// TwinCAT 3 PLC project Tc3EventLoggerListener
// Title: Tc3EventLoggerListener
// Company: tchaxx
// Author: densogiaichned
// ProjectVersion: 0.0.1.0
// Description: Example how to use TC3 EventLogger
// ProgramVersion: 3.1.4024.0
// libraries:
//   Tc2_Standard, * (Beckhoff Automation GmbH)
//   Tc2_System, * (Beckhoff Automation GmbH)
//   Tc2_Utilities, * (Beckhoff Automation GmbH)
//   Tc3_EventLogger, * (Beckhoff Automation GmbH)
//   Tc3_Module, * (Beckhoff Automation GmbH)
//   TcUnit, * (www.tcunit.org)
// project tree:
//   DUTs/ E_EventLoggerListenerState.TcTLEO, E_LanguageId.TcTLEO, ST_LoggedEvent.TcDUT, ST_RequestEventTexts.TcDUT, T_LoggedEvents.TcDUT, T_RequestEventTexts.TcDUT
//   GVLs/ Param_EventLoggerListener.TcGVL
//   ITFs/ I_LoggedEventsSort.TcIO
//   / PlcTask.TcTTO, PlcTaskUnitTest.TcTTO
//   POUs/ FB_EventLoggerListenerImpl.TcPOU, FB_LoggedEventsSortAscending.TcPOU, FB_LoggedEventsSortDescending.TcPOU, MAIN.TcPOU
//   TESTs/ FB_LoggedEventsSortDescending_Tests.TcPOU, PRG_UnitTests.TcPOU
// real-time tasks:
//   TASK PlcTask: cycle T#10ms, priority 20, ADS port 350
//   TASK PlcTaskUnitTest: cycle T#10ms, priority 1, ADS port 351

CONFIGURATION Tc3EventLoggerListener
    RESOURCE PLC ON TwinCAT3
        TASK PlcTask(INTERVAL := T#10ms, PRIORITY := 20);
        TASK PlcTaskUnitTest(INTERVAL := T#10ms, PRIORITY := 1);
        PROGRAM MAIN WITH PlcTask : MAIN;
        PROGRAM PRG_UnitTests WITH PlcTaskUnitTest : PRG_UnitTests;
    END_RESOURCE
END_CONFIGURATION

// ---- DUTs/E_EventLoggerListenerState.TcTLEO
{attribute 'qualified_only'}
{attribute 'strict'}
{attribute 'to_string'}
TYPE E_EventLoggerListenerState :
(	 
	eIdle := 0,
	eInit:= 1, 
	eListening:= 10, 
	eRetrieveTexts:= 20,
	eSortEvents := 30,
	eDone := 100,
	eError := -1
);
END_TYPE
//  eError = '-1'

// ---- DUTs/E_LanguageId.TcTLEO
{attribute 'qualified_only'}
{attribute 'strict'}
TYPE E_LanguageId :
(
	ar_SA := 1025 , // Arabic - Saudi Arabia
	bg_BG := 1026 , // Bulgarian
	ca_ES := 1027 , // Catalan
	zh_TW := 1028 , // Chinese - Taiwan
	cs_CZ := 1029 , // Czech
	da_DK := 1030 , // Danish
	de_DE := 1031 , // German - Germany
	el_GR := 1032 , // Greek
	en_US := 1033 , // English - United States
	es_ES := 1034 , // Spanish - Spain (Traditional Sort)
	fi_FI := 1035 , // Finnish
	fr_FR := 1036 , // French - France
	he_IL := 1037 , // Hebrew
	hu_HU := 1038 , // Hungarian
	is_IS := 1039 , // Icelandic
	it_IT := 1040 , // Italian - Italy
	ja_JP := 1041 , // Japanese
	ko_KR := 1042 , // Korean
	nl_NL := 1043 , // Dutch - Netherlands
	nb_NO := 1044 , // Norwegian (Bokmål)
	pl_PL := 1045 , // Polish
	pt_BR := 1046 , // Portuguese - Brazil
	rm_CH := 1047 , // Rhaeto-Romanic
	ro_RO := 1048 , // Romanian
	ru_RU := 1049 , // Russian
	hr_HR := 1050 , // Croatian
	sk_SK := 1051 , // Slovak
	sq_AL := 1052 , // Albanian - Albania
	sv_SE := 1053 , // Swedish
	th_TH := 1054 , // Thai
	tr_TR := 1055 , // Turkish
	ur_PK := 1056 , // Urdu - Pakistan
	id_ID := 1057 , // Indonesian
	uk_UA := 1058 , // Ukrainian
	be_BY := 1059 , // Belarusian
	sl_SI := 1060 , // Slovenian
	et_EE := 1061 , // Estonian
	lv_LV := 1062 , // Latvian
	lt_LT := 1063 , // Lithuanian
	tg_Cyrl_TJ := 1064 , // Tajik
	fa_IR := 1065 , // Persian
	vi_VN := 1066 , // Vietnamese
	hy_AM := 1067 , // Armenian - Armenia
	az_Latn_AZ := 1068 , // Azerbaijani (Latin)
	eu_ES := 1069 , // Basque
	wen_DE := 1070 , // Sorbian
	mk_MK := 1071 , // North Macedonian
	st_ZA := 1072 , // Sutu
	ts_ZA := 1073 , // Tsonga
	tn_ZA := 1074 , // Tswana
	ven_ZA := 1075 , // Venda
	xh_ZA := 1076 , // Xhosa
	zu_ZA := 1077 , // Zulu
	af_ZA := 1078 , // Afrikaans - South Africa
	ka_GE := 1079 , // Georgian
	fo_FO := 1080 , // Faroese
	hi_IN := 1081 , // Hindi
	mt_MT := 1082 , // Maltese
	se_NO := 1083 , // Sami
	gd_GB := 1084 , // Scottish Gaelic
	yi := 1085 , // Yiddish
	ms_MY := 1086 , // Malay - Malaysia
	kk_KZ := 1087 , // Kazakh
	ky_KG := 1088 , // Kyrgyz (Cyrillic)
	sw_KE := 1089 , // Swahili
	tk_TM := 1090 , // Turkmen
	uz_Latn_UZ := 1091 , // Uzbek (Latin)
	tt_RU := 1092 , // Tatar
	bn_IN := 1093 , // Bengali (India)
	pa_IN := 1094 , // Punjabi
	gu_IN := 1095 , // Gujarati
	or_IN := 1096 , // Odia
	ta_IN := 1097 , // Tamil
	te_IN := 1098 , // Telugu
	kn_IN := 1099 , // Kannada
	ml_IN := 1100 , // Malayalam
	as_IN := 1101 , // Assamese
	mr_IN := 1102 , // Marathi
	sa_IN := 1103 , // Sanskrit
	mn_MN := 1104 , // Mongolian (Cyrillic)
	bo_CN := 1105 , // Tibetan - People's Republic of China
	cy_GB := 1106 , // Welsh
	km_KH := 1107 , // Khmer
	lo_LA := 1108 , // Lao
	my_MM := 1109 , // Burmese
	gl_ES := 1110 , // Galician
	kok_IN := 1111 , // Konkani
	mni := 1112 , // Manipuri
	sd_IN := 1113 , // Sindhi - India
	syr_SY := 1114 , // Syriac
	si_LK := 1115 , // Sinhalese - Sri Lanka
	chr_US := 1116 , // Cherokee - United States
	iu_Cans_CA := 1117 , // Inuktitut
	am_ET := 1118 , // Amharic - Ethiopia
	tmz := 1119 , // Tamazight (Arabic)
	ks_Arab_IN := 1120 , // Kashmiri (Arabic)
	ne_NP := 1121 , // Nepali
	fy_NL := 1122 , // Frisian - Netherlands
	ps_AF := 1123 , // Pashto
	fil_PH := 1124 , // Filipino
	dv_MV := 1125 , // Divehi
	bin_NG := 1126 , // Edo
	fuv_NG := 1127 , // Fulfulde - Nigeria
	ha_Latn_NG := 1128 , // Hausa - Nigeria
	ibb_NG := 1129 , // Ibibio - Nigeria
	yo_NG := 1130 , // Yoruba
	quz_BO := 1131 , // Quecha - Bolivia
	nso_ZA := 1132 , // Sepedi
	ig_NG := 1136 , // Igbo - Nigeria
	kr_NG := 1137 , // Kanuri - Nigeria
	gaz_ET := 1138 , // Oromo
	ti_ER := 1139 , // Tigrigna - Ethiopia
	gn_PY := 1140 , // Guarani - Paraguay
	haw_US := 1141 , // Hawaiian - United States
	la := 1142 , // Latin
	so_SO := 1143 , // Somali
	ii_CN := 1144 , // Yi
	pap_AN := 1145 , // Papiamentu
	ug_Arab_CN := 1152 , // Uighur - China
	mi_NZ := 1153 , // Maori - New Zealand
	ar_IQ := 2049 , // Arabic - Iraq
	zh_CN := 2052 , // Chinese - People's Republic of China
	de_CH := 2055 , // German - Switzerland
	en_GB := 2057 , // English - United Kingdom
	es_MX := 2058 , // Spanish - Mexico
	fr_BE := 2060 , // French - Belgium
	it_CH := 2064 , // Italian - Switzerland
	nl_BE := 2067 , // Dutch - Belgium
	nn_NO := 2068 , // Norwegian (Nynorsk)
	pt_PT := 2070 , // Portuguese - Portugal
	ro_MD := 2072 , // Romanian - Moldova
	ru_MD := 2073 , // Russian - Moldava
	sr_Latn_CS := 2074 , // Serbian (Latin)
	sv_FI := 2077 , // Swedish - Finland
	ur_IN := 2080 , // Urdu - India
	az_Cyrl_AZ := 2092 , // Azerbaijani (Cyrillic)
	ga_IE := 2108 , // Irish
	ms_BN := 2110 , // Malay - Brunei Darussalam
	uz_Cyrl_UZ := 2115 , // Uzbek (Cyrillic)
	bn_BD := 2117 , // Bangla
	pa_PK := 2118 , // Punjabi (Pakistan)
	mn_Mong_CN := 2128 , // Mongolian (Mongolian)
	bo_BT := 2129 , // Tibetan - Bhutan
	sd_PK := 2137 , // Sindhi - Pakistan
	tzm_Latn_DZ := 2143 , // Tamazight (Latin)
	ks_Deva_IN := 2144 , // Kashmiri (Devanagari)
	ne_IN := 2145 , // Nepali - India
	quz_EC := 2155 , // Quecha - Ecuador
	ti_ET := 2163 , // Tigrigna - Eritrea
	ar_EG := 3073 , // Arabic - Egypt
	zh_HK := 3076 , // Chinese - Hong Kong SAR
	de_AT := 3079 , // German - Austria
	en_AU := 3081 , // English - Australia
	es_ES2 := 3082 , // Spanish - Spain (Modern Sort)
	fr_CA := 3084 , // French - Canada
	sr_Cyrl_CS := 3098 , // Serbian (Cyrillic)
	quz_PE := 3179 , // Quecha - Peru
	ar_LY := 4097 , // Arabic - Libya
	zh_SG := 4100 , // Chinese - Singapore
	de_LU := 4103 , // German - Luxembourg
	en_CA := 4105 , // English - Canada
	es_GT := 4106 , // Spanish - Guatemala
	fr_CH := 4108 , // French - Switzerland
	hr_BA := 4122 , // Croatian (Bosnia/Herzegovina)
	ar_DZ := 5121 , // Arabic - Algeria
	zh_MO := 5124 , // Chinese - Macao SAR
	de_LI := 5127 , // German - Liechtenstein
	en_NZ := 5129 , // English - New Zealand
	es_CR := 5130 , // Spanish - Costa Rica
	fr_LU := 5132 , // French - Luxembourg
	bs_Latn_BA := 5146 , // Bosnian (Bosnia/Herzegovina)
	ar_MO := 6145 , // Arabic - Morocco
	en_IE := 6153 , // English - Ireland
	es_PA := 6154 , // Spanish - Panama
	fr_MC := 6156 , // French - Monaco
	ar_TN := 7169 , // Arabic - Tunisia
	en_ZA := 7177 , // English - South Africa
	es_DO := 7178 , // Spanish - Dominican Republic
	ar_OM := 7180 , // French - West Indies,fr-Arabic - Oman
	en_JM := 8201 , // English - Jamaica
	es_VE := 8202 , // Spanish - Venezuela
	fr_RE := 8204 , // French - Reunion
	ar_YE := 9217 , // Arabic - Yemen
	es_CO := 9225 , // English - Caribbean,en-Spanish - Colombia
	fr_CG := 9228 , // French - Democratic Rep. of Congo
	ar_SY := 10241 , // Arabic - Syria
	en_BZ := 10249 , // English - Belize
	es_PE := 10250 , // Spanish - Peru
	fr_SN := 10252 , // French - Senegal
	ar_JO := 11265 , // Arabic - Jordan
	en_TT := 11273 , // English - Trinidad
	es_AR := 11274 , // Spanish - Argentina
	fr_CM := 11276 , // French - Cameroon
	ar_LB := 12289 , // Arabic - Lebanon
	en_ZW := 12297 , // English - Zimbabwe
	es_EC := 12298 , // Spanish - Ecuador
	fr_CI := 12300 , // French - Cote d'Ivoire
	ar_KW := 13313 , // Arabic - Kuwait
	en_PH := 13321 , // English - Philippines
	es_CL := 13322 , // Spanish - Chile
	fr_ML := 13324 , // French - Mali
	ar_AE := 14337 , // Arabic - U.A.E.
	en_ID := 14345 , // English - Indonesia
	es_UY := 14346 , // Spanish - Uruguay
	fr_MA := 14348 , // French - Morocco
	ar_BH := 15361 , // Arabic - Bahrain
	en_HK := 15369 , // English - Hong Kong SAR
	es_PY := 15370 , // Spanish - Paraguay
	fr_HT := 15372 , // French - Haiti
	ar_QA := 16385 , // Arabic - Qatar
	en_IN := 16393 , // English - India
	es_BO := 16394 , // Spanish - Bolivia
	en_MY := 17417 , // English - Malaysia
	es_SV := 17418 , // Spanish - El Salvador
	en_SG := 18441 , // English - Singapore
	es_HN := 18442 , // Spanish - Honduras
	es_NI := 19466 , // Spanish - Nicaragua
	es_PR := 20490 , // Spanish - Puerto Rico
	es_US := 21514 , // Spanish - United States
	es_419 := 58378, // Spanish - Latin Americaa
	fr_015 := 58380  // French - North Africa
);
END_TYPE

// ---- DUTs/ST_LoggedEvent.TcDUT
TYPE ST_LoggedEvent :
STRUCT
	EventClass			: GUID;
	sEventClassName		: STRING(Param_EventLoggerListener.cEventClassNameLength);
	nEventId			: UDINT;
	nUniqueId			: UDINT;
	eSeverity			: TcEventSeverity;
	sMessageText 		: STRING(Param_EventLoggerListener.cMessageTextLength);
	sSourceName 		: STRING(Param_EventLoggerListener.cMessageTextLength);
	nSourceId			: UDINT;
	nTimestampRaised 	: ULINT;	
	nTimestampConfirmed	: ULINT;
	nTimestampCleared 	: ULINT;
	sJson				: STRING (Param_EventLoggerListener.cMaxJsonTextLength);
END_STRUCT
END_TYPE

// ---- DUTs/ST_RequestEventTexts.TcDUT
TYPE ST_RequestEventTexts :
STRUCT
	fbEventText 		: FB_RequestEventText;
	fbEventClassName 	: FB_RequestEventClassName;
	bAssigned			: BOOL;
	bReqEventText		: BOOL;
	bReqClassName		: BOOL;
	nIndex				: UDINT;
END_STRUCT
END_TYPE

// ---- DUTs/T_LoggedEvents.TcDUT
TYPE T_LoggedEvents : 
	ARRAY[0..Param_EventLoggerListener.cMaxConcurrentEvents - 1] OF ST_LoggedEvent; 
END_TYPE

// ---- DUTs/T_RequestEventTexts.TcDUT
TYPE T_RequestEventTexts : 
	ARRAY[0..Param_EventLoggerListener.cMaxConcurrentEvents - 1] OF ST_RequestEventTexts; 
END_TYPE

// ---- GVLs/Param_EventLoggerListener.TcGVL
{attribute 'qualified_only'}
VAR_GLOBAL CONSTANT
	cEventClassNameLength : UDINT (80..255) := 80;
	cMessageTextLength : UDINT(80..1024) := 255;
	cSourceNameLength : UDINT (80..255) := 80;
	cMaxConcurrentEvents : UDINT (1..64) := 16;
	cMaxJsonTextLength : UDINT (80..16384) := 1024;
END_VAR

// ---- ITFs/I_LoggedEventsSort.TcIO
INTERFACE I_LoggedEventsSort

METHOD Sort : HRESULT
VAR_IN_OUT
	aLoggedEvents : T_LoggedEvents;
END_VAR
END_METHOD

END_INTERFACE

// ---- POUs/MAIN.TcPOU
PROGRAM MAIN
VAR
	fbEventLoggerListener 	: FB_EventLoggerListenerImpl;
	aLoggedEvents 			: T_LoggedEvents;
	
	fbSortAscending			: FB_LoggedEventsSortAscending;
	fbSortDescending		: FB_LoggedEventsSortDescending;
END_VAR


fbEventLoggerListener(aLoggedEvents:= aLoggedEvents, ipSort:= fbSortDescending);

END_PROGRAM

// ---- POUs/FB_EventLoggerListenerImpl.TcPOU
{attribute 'reflection'}
FUNCTION_BLOCK FB_EventLoggerListenerImpl EXTENDS FB_ListenerBase2
VAR_INPUT
	bEnable				: BOOL;
	eLanguageId			: E_LanguageId := E_LanguageId.en_US;
	ipSort				: I_LoggedEventsSort := NULL;
END_VAR
VAR_IN_OUT
	aLoggedEvents 		:	T_LoggedEvents;
END_VAR
VAR_OUTPUT
	bBusy				: BOOL;
	bDone				: BOOL;
	bError				: BOOL;
	nErrorCode			: DINT;
	nReceivedEvents		: UDINT;
END_VAR
VAR_INPUT
	ipEventFilter 		: I_TcEventFilterBase; //OPTIONAL: Pointer to an instance of FB_TcEventFilter, if a filter is to be activated. Otherwise, listening to ALL events.
END_VAR
VAR_OUTPUT
END_VAR

VAR
	fbDefaultFilter 	: FB_TcEventFilter;
	pEventToProcess		: POINTER TO ST_LoggedEvent := NULL;
	aRequestEventTexts 	: T_RequestEventTexts;
	refLoggedEvents 	: REFERENCE TO T_LoggedEvents;	// Prevents warning "Access to VAR_IN_OUT from external context"
END_VAR

VAR
	hr 					: HRESULT;
END_VAR

VAR CONSTANT
	cUpperBound			: UDINT := Param_EventLoggerListener.cMaxConcurrentEvents - 1;
END_VAR

VAR
	{attribute 'hide'}
	eEventState 		: E_EventLoggerListenerState := E_EventLoggerListenerState.eInit;
	{attribute 'hide'}
    {attribute 'instance-path'} 
    {attribute 'noinit'} 
	sInstancePath		: STRING;
END_VAR

refLoggedEvents REF= aLoggedEvents;

IF NOT bEnable THEN
	eEventLoggerListenerState := E_EventLoggerListenerState.eIdle;
END_IF

CASE eEventLoggerListenerState OF
	
	E_EventLoggerListenerState.eIdle:
		hr := Idle();
		ActivateStateOrError(hr, eNextState:= E_EventLoggerListenerState.eInit); 
		
	E_EventLoggerListenerState.eInit:		
		hr := Init(aLoggedEvents);
		IF FAILED(hr) THEN
			eEventLoggerListenerState := E_EventLoggerListenerState.eError;
		ELSE
			eEventLoggerListenerState := E_EventLoggerListenerState.eListening;
		END_IF
		
	E_EventLoggerListenerState.eListening:
		hr := Listening();
		IF FAILED(hr) THEN
			eEventLoggerListenerState := E_EventLoggerListenerState.eError;
		ELSIF HasReceivedEvents() THEN
			eEventLoggerListenerState := E_EventLoggerListenerState.eRetrieveTexts;
		END_IF
				
	E_EventLoggerListenerState.eRetrieveTexts:
		hr := RetrieveTexts(aLoggedEvents);
		ActivateStateOrError(hr, eNextState:= E_EventLoggerListenerState.eSortEvents);
		
	E_EventLoggerListenerState.eSortEvents:
		hr := SortEvents();
		IF FAILED(hr) THEN
			eEventLoggerListenerState := E_EventLoggerListenerState.eError;
		ELSE
			eEventLoggerListenerState := E_EventLoggerListenerState.eDone;
		END_IF
	
	E_EventLoggerListenerState.eDone:
		Done();
		
	E_EventLoggerListenerState.eError:
		Error(hr);
		
END_CASE

bError 	:= eEventLoggerListenerState = E_EventLoggerListenerState.eError; 
bBusy 	:= bEnable AND NOT bError AND NOT (eEventLoggerListenerState = E_EventLoggerListenerState.eDone); 
bDone	:= eEventLoggerListenerState = E_EventLoggerListenerState.eDone;

METHOD PRIVATE ActivateStateOrError : BOOL
VAR_INPUT
	hr 			: HRESULT;
	eNextState 	: E_EventLoggerListenerState;
END_VAR
ActivateStateOrError := TRUE;
IF FAILED(hr) THEN
	eEventLoggerListenerState := E_EventLoggerListenerState.eError;
ELSIF hr = S_OK THEN
	eEventLoggerListenerState := eNextState;
ELSE 
	// other results, e.g. S_PENDING, S_FALSE
	ActivateStateOrError := FALSE;
END_IF
END_METHOD

METHOD PRIVATE ClearEventBuffer
VAR_IN_OUT
	aEventsBuffer 	: T_LoggedEvents;
	aReqEventTexts 	: T_RequestEventTexts;
END_VAR
VAR
	i : UDINT;
END_VAR
nReceivedEvents := 0;
FOR i := 0 TO cUpperBound DO 	
	MEMSET(destAddr:= ADR(aEventsBuffer[i]), 16#0, SIZEOF(aEventsBuffer[i]));
	aReqEventTexts[i].bAssigned := FALSE;
	aReqEventTexts[i].bReqEventText := FALSE;
	aReqEventTexts[i].bReqClassName := FALSE;
	aReqEventTexts[i].nIndex := 0;
END_FOR
END_METHOD

METHOD PRIVATE Done : HRESULT
VAR_INPUT
END_VAR
Done := S_OK;
END_METHOD

PROPERTY PRIVATE eEventLoggerListenerState : E_EventLoggerListenerState
GET
eEventLoggerListenerState := eEventState;
END_GET
SET
VAR
	sStateOld : STRING;
END_VAR

VAR_INST
	fbFrmt : FB_FormatString2;
	sErrorMessage : T_MaxString;
END_VAR

VAR CONSTANT
	cErrorFrmt : STRING := '[%s] Error in step $'%s$': hr=0x%08X';
END_VAR
 
IF eEventState <> eEventLoggerListenerState AND_THEN eEventLoggerListenerState = E_EventLoggerListenerState.eError THEN
	sStateOld := TO_STRING(eEventState);	
	fbFrmt(
	pFormatString:= ADR(cErrorFrmt) , 
	arg1:= F_STRINGEx(sInstancePath),
	arg2:= F_STRINGEx(sStateOld), 
	arg3:= F_DINT(hr), 
	pDstString:= ADR(sErrorMessage), 
	nDstSize:= SIZEOF(sErrorMessage) -1 );
	ADSLOGSTR(msgCtrlMask:= ADSLOG_MSGTYPE_ERROR, msgFmtStr:= '%s', strArg:= sErrorMessage);
END_IF

eEventState := eEventLoggerListenerState;
END_SET
END_PROPERTY

METHOD PRIVATE Error
VAR_INPUT
	hr : HRESULT;
END_VAR
nErrorCode := hr;
END_METHOD

METHOD PRIVATE GetEventTexts : HRESULT
VAR_IN_OUT
	aLoggedEvents  : T_LoggedEvents;
	aReqEventTexts : T_RequestEventTexts;
END_VAR
VAR
	i				: UDINT;
	hr				: HRESULT;
	refReqEventText : REFERENCE TO ST_RequestEventTexts;
	refLoggedEvent 	: REFERENCE TO ST_LoggedEvent;
	
	bEventDone, bClassNameDone : BOOL;
	bEventError, bClassNameError : BOOL;
END_VAR

GetEventTexts := S_OK;

FOR i := 0 TO cUpperBound DO
	
	refReqEventText REF= aReqEventTexts[i];	
	IF NOT refReqEventText.bAssigned THEN
		CONTINUE;
	END_IF
	
	refLoggedEvent 	REF= aLoggedEvents[refReqEventText.nIndex];
	
	bEventDone 		:= refReqEventText.bAssigned AND (NOT refReqEventText.fbEventText.bBusy AND NOT refReqEventText.fbEventText.bError);
	bClassNameDone 	:= refReqEventText.bAssigned AND (NOT refReqEventText.fbEventClassName.bBusy AND NOT refReqEventText.fbEventClassName.bError);
	
	IF bEventDone AND refReqEventText.bReqEventText THEN
		refReqEventText.fbEventText.GetString(refLoggedEvent.sMessageText, SIZEOF(refLoggedEvent.sMessageText) - 1);
		refReqEventText.bReqEventText := FALSE;		
	END_IF
	
	IF bClassNameDone AND refReqEventText.bReqClassName THEN
		refReqEventText.fbEventClassName.GetString(refLoggedEvent.sEventClassName, SIZEOF(refLoggedEvent.sEventClassName) - 1);
		refReqEventText.bReqClassName := FALSE;
	END_IF
	
	bEventError		:= refReqEventText.bAssigned AND refReqEventText.bReqEventText AND refReqEventText.fbEventText.bError;
	bClassNameError	:= refReqEventText.bAssigned AND refReqEventText.bReqClassName AND refReqEventText.fbEventClassName.bError;
	
	IF bEventError THEN
		hr := refReqEventText.fbEventText.hrErrorCode;
		refLoggedEvent.sMessageText := RequestEventTextsError(sFrmt:= 'Couldn$'t get EventText: hr=0x%08X', F_DINT(hr));	
		refReqEventText.bReqEventText := FALSE;	
	END_IF
	
	IF bClassNameError THEN
		hr := refReqEventText.fbEventClassName.hrErrorCode;
		refLoggedEvent.sEventClassName := RequestEventTextsError(sFrmt:= 'Couldn$'t get ClassName: hr=0x%08X', F_DINT(hr));	
		refReqEventText.bReqClassName := FALSE;
	END_IF
	
	IF refReqEventText.bAssigned AND (refReqEventText.bReqEventText OR_ELSE refReqEventText.bReqClassName) THEN
		GetEventTexts := S_PENDING;
	END_IF
	
END_FOR
END_METHOD

METHOD PRIVATE HasReceivedEvents : BOOL
VAR
	i : UDINT;
END_VAR
FOR i := 0 TO cUpperBound DO
	IF THIS^.aRequestEventTexts[i].bAssigned THEN 
		HasReceivedEvents := TRUE;
		RETURN;
	END_IF
END_FOR
END_METHOD

METHOD PRIVATE Idle : HRESULT
VAR_INPUT
END_VAR
Idle := S_PENDING;

IF bEnable THEN
	Idle := S_OK;
END_IF
END_METHOD

METHOD PRIVATE Init : HRESULT
VAR_IN_OUT
	aLoggedEvents 		:	T_LoggedEvents;
END_VAR
ClearEventBuffer(aEventsBuffer:= aLoggedEvents, aReqEventTexts:= aRequestEventTexts);
Init := Setup(ipEventFilter);
END_METHOD

METHOD PRIVATE Listening : HRESULT
VAR_INPUT
END_VAR
Listening := SUPER^.Execute();
END_METHOD

METHOD OnAlarmCleared : HRESULT
VAR_INPUT
	fbEvent : REFERENCE TO FB_TcEvent;
END_VAR

VAR
	stLoggedEvent : ST_LoggedEvent;
END_VAR
stLoggedEvent := To_StLoggedEvent(fbEvent);
stLoggedEvent.nTimestampRaised := 0;
stLoggedEvent.nTimestampCleared := fbEvent.nTimestamp;

OnAlarmCleared := StoreEvent(stLoggedEvent, fbEvent);
END_METHOD

METHOD OnAlarmConfirmed : HRESULT
VAR_INPUT
	fbEvent : REFERENCE TO FB_TcEvent;
END_VAR

VAR
	stLoggedEvent 	: ST_LoggedEvent;
	bNoMoreEvents 	: BOOL;
	hr 				: HRESULT;
END_VAR
stLoggedEvent := To_StLoggedEvent(fbEvent);
stLoggedEvent.nTimestampRaised := 0;
stLoggedEvent.nTimestampConfirmed := fbEvent.nTimestamp;

OnAlarmConfirmed := StoreEvent(stLoggedEvent, fbEvent);
END_METHOD

METHOD OnAlarmRaised : HRESULT
VAR_INPUT
	fbEvent : REFERENCE TO FB_TcEvent;
END_VAR

VAR
	stLoggedEvent 	: ST_LoggedEvent;
	bNoMoreEvents 	: BOOL;
	refReqEventText : REFERENCE TO ST_RequestEventTexts;
	nIndex 			: UDINT;
END_VAR
stLoggedEvent := To_StLoggedEvent(fbEvent);
stLoggedEvent.nTimestampRaised := fbEvent.nTimestamp;

OnAlarmRaised := StoreEvent(stLoggedEvent, fbEvent);
END_METHOD

METHOD OnMessageSent : HRESULT
VAR_INPUT
	fbEvent : REFERENCE TO FB_TcEvent;
END_VAR

VAR
	stLoggedEvent 	: ST_LoggedEvent;
	bNoMoreEvents 	: BOOL;
	refReqEventText : REFERENCE TO ST_RequestEventTexts;
	nIndex 			: UDINT;
END_VAR
stLoggedEvent := To_StLoggedEvent(fbEvent);
OnMessageSent := StoreEvent(stLoggedEvent, fbEvent);
END_METHOD

METHOD PRIVATE RequestEventTextsError : STRING(Param_EventLoggerListener.cMessageTextLength)
VAR_IN_OUT CONSTANT
	sFrmt : STRING;
END_VAR
VAR_INPUT
	tArg  : T_ARG;	
END_VAR
VAR_INST
	fbFrmt		: FB_FormatString2;
END_VAR


fbFrmt(
	pFormatString:= ADR(sFrmt), 
	arg1:= tArg,  
	pDstString:= ADR(RequestEventTextsError), 
	nDstSize:= SIZEOF(RequestEventTextsError) - 1, 
	bError=> , 
	nErrId=> );
END_METHOD

METHOD PRIVATE RetrieveTexts : HRESULT
VAR_IN_OUT
	aLoggedEvents 		:	T_LoggedEvents;
END_VAR
{warning 'TODO: Timeout ?!'}

hr := GetEventTexts(aReqEventTexts:= aRequestEventTexts, aLoggedEvents:= aLoggedEvents);
END_METHOD

METHOD PRIVATE Setup : HRESULT
VAR_INPUT
	ipEventFilter 	: I_TcEventFilterBase;
END_VAR

VAR
	hr : HRESULT;
END_VAR


VAR_INST
	ipEventFilterInUse	: I_TcEventFilterBase;
END_VAR
IF ipEventFilterInUse <> NULL AND_THEN (ipEventFilter = NULL OR_ELSE ipEventFilter = ipEventFilterInUse) THEN
	Setup := S_FALSE;
	RETURN;
END_IF

IF ipEventFilterInUse <> NULL  AND_THEN ipEventFilter <> ipEventFilterInUse THEN
	SUPER^.Unsubscribe();
END_IF

IF ipEventFilter <> NULL THEN	
	hr := SUPER^.Subscribe2(ipEventFilter);
	ipEventFilterInUse := ipEventFilter;
ELSE
	fbDefaultFilter.Clear().EventId.GreaterThan(0);
	hr := SUPER^.Subscribe2(ipEventFilter:= fbDefaultFilter);
	ipEventFilterInUse := fbDefaultFilter;
END_IF

Setup := hr;
END_METHOD

METHOD PRIVATE SortEvents : HRESULT
VAR_INPUT
END_VAR


IF ipSort = NULL THEN
	SortEvents := S_OK;
	RETURN;
END_IF

IF NOT __ISVALIDREF(refLoggedEvents) THEN
	SortEvents := E_FAIL;
	RETURN;
END_IF;

SortEvents := ipSort.Sort(aLoggedEvents:= refLoggedEvents);
END_METHOD

METHOD PRIVATE StoreEvent : HRESULT
VAR_INPUT CONSTANT
	stLoggedEvent 	: REFERENCE TO ST_LoggedEvent;
	fbEvent			: REFERENCE TO FB_TcEvent;
END_VAR

VAR
	i : UDINT;
	refReqEventText : REFERENCE TO ST_RequestEventTexts;
END_VAR

IF NOT __ISVALIDREF(refLoggedEvents) THEN
	StoreEvent := E_FAIL;
	RETURN;
END_IF;	

FOR i := 0 TO cUpperBound  DO
	IF NOT THIS^.aRequestEventTexts[i].bAssigned THEN
		
	
		refLoggedEvents[i] := stLoggedEvent;
		
		refReqEventText REF= THIS^.aRequestEventTexts[i];
		refReqEventText.nIndex := i;
		refReqEventText.bAssigned := TRUE;
		refReqEventText.fbEventText.Clear();
		refReqEventText.fbEventText.Request(eventClass:= fbEvent.EventClass, nEventId:= fbEvent.nEventId, nLangId:= eLanguageId, ipArgs:= fbEvent.ipArguments);
		refReqEventText.bReqEventText := TRUE;
		refReqEventText.fbEventClassName.Clear();
		refReqEventText.fbEventClassName.Request(eventClass:= fbEvent.EventClass, nLangId:= eLanguageId);
		refReqEventText.bReqClassName := TRUE;
		
		nReceivedEvents := nReceivedEvents + 1;
		EXIT;
	END_IF; 
END_FOR

IF THIS^.aRequestEventTexts[cUpperBound].bAssigned THEN
	StoreEvent := S_PENDING;
ELSE
	StoreEVent := S_OK;
END_IF
END_METHOD

METHOD PRIVATE To_StLoggedEvent : ST_LoggedEvent
VAR_INPUT CONSTANT
	fbEvent : REFERENCE TO FB_TcEvent;
END_VAR
To_StLoggedEvent.nEventId			:= fbEvent.nEventId;
To_StLoggedEvent.nSourceId			:= fbEvent.ipSourceInfo.nId;
To_StLoggedEvent.sSourceName		:= fbEvent.ipSourceInfo.sName;
To_StLoggedEvent.eSeverity 			:= fbEvent.eSeverity;
To_StLoggedEvent.EventClass 		:= fbEvent.EventClass;
To_StLoggedEvent.nTimestampRaised	:= fbEvent.nTimestamp;
To_StLoggedEvent.nUniqueId 			:= fbEvent.nUniqueId;

fbEvent.GetJsonAttribute(To_StLoggedEvent.sJson, SIZEOF(To_StLoggedEvent.sJson) - 1);
END_METHOD

END_FUNCTION_BLOCK

// ---- POUs/FB_LoggedEventsSortAscending.TcPOU
{attribute 'no_explicit_call' := 'do not call this POU directly'}
FUNCTION_BLOCK FINAL FB_LoggedEventsSortAscending IMPLEMENTS I_LoggedEventsSort
VAR_INPUT
END_VAR
VAR_OUTPUT
END_VAR
VAR
END_VAR

METHOD Sort : HRESULT
VAR_IN_OUT
	aLoggedEvents	: T_LoggedEvents;
END_VAR
{warning 'TODO: Implement sorting in ascending order'}
Sort := S_OK;
END_METHOD

END_FUNCTION_BLOCK

// ---- POUs/FB_LoggedEventsSortDescending.TcPOU
{attribute 'no_explicit_call' := 'do not call this POU directly'}
FUNCTION_BLOCK FINAL FB_LoggedEventsSortDescending IMPLEMENTS I_LoggedEventsSort
VAR_INPUT
END_VAR
VAR_OUTPUT
END_VAR
VAR
END_VAR

METHOD PRIVATE GetLastIndex : UDINT
VAR_IN_OUT
	aLoggedEvents	: T_LoggedEvents;
END_VAR

VAR
	i 				: UDINT;
	nLastIndex		: UDINT;
	stLoggedEvent 	: ST_LoggedEvent;
END_VAR
FOR i := 0 TO Param_EventLoggerListener.cMaxConcurrentEvents - 1 BY 1 DO
	IF aLoggedEvents[i].nUniqueId > 0 OR_ELSE aLoggedEvents[i].nSourceId > 0 THEN
		GetLastIndex := i;
	ELSE
		EXIT;
	END_IF
END_FOR;
END_METHOD

METHOD Sort : HRESULT
VAR_IN_OUT
	aLoggedEvents	: T_LoggedEvents;
END_VAR

VAR
	i 				: UDINT;
	nLastIndex		: UDINT;
	stTmpEvent 		: ST_LoggedEvent;
END_VAR
nLastIndex := GetLastIndex(aLoggedEvents);
IF nLastIndex = 0 THEN
	Sort := S_FALSE;
	RETURN;
END_IF

FOR i := nLastIndex TO (nLastIndex / 2) + 1 BY -1 DO
	MEMMOVE(destAddr:= ADR(stTmpEvent), srcAddr:= ADR(aLoggedEvents[i]), n:= SIZEOF(stTmpEvent)); 
	MEMMOVE(destAddr:= ADR(aLoggedEvents[i]), srcAddr:= ADR(aLoggedEvents[nLastIndex - i]), n:= SIZEOF(aLoggedEvents[i])); 
	MEMMOVE(destAddr:= ADR(aLoggedEvents[nLastIndex - i]), srcAddr:= ADR(stTmpEvent), n:= SIZEOF(stTmpEvent)); 
END_FOR

Sort := S_OK;
END_METHOD

END_FUNCTION_BLOCK

// ---- TESTs/PRG_UnitTests.TcPOU
{attribute 'analysis' := '-33'}
PROGRAM PRG_UnitTests

VAR
{IF defined (UNIT_TEST)}	
	fbLoggedEventsSortDescendingTests : FB_LoggedEventsSortDescending_Tests;
{END_IF}
END_VAR

{IF defined (UNIT_TEST)}

TcUnit.RUN();

{END_IF}

END_PROGRAM

// ---- TESTs/FB_LoggedEventsSortDescending_Tests.TcPOU
{attribute 'reflection'}
FUNCTION_BLOCK FINAL FB_LoggedEventsSortDescending_Tests EXTENDS TcUnit.FB_TestSuite
VAR_INPUT
END_VAR
VAR_OUTPUT
END_VAR
VAR
	{attribute 'instance-path'} 
    {attribute 'noinit'} 
	sTestName			: T_MaxString;

END_VAR


TEST(sTestName);

ShouldDoNothingWhenEmpty();
ShouldDoNothingIfOnlyOneEvent();
ShouldSortTwoEventsInDescendingOrderSuccessfully();
ShouldSortThreeEventsInDescendingOrderSuccessfully();
ShouldSortFourEventsInDescendingOrderSuccessfully();
ShouldSortFiveEventsInDescendingOrderSuccessfully();
ShouldSortXEventsInDescendingOrderSuccessfully();
TEST_FINISHED_NAMED(sTestName);

METHOD PRIVATE ShouldDoNothingIfOnlyOneEvent
VAR_INPUT
END_VAR
VAR_INST
	fbSUT	: FB_LoggedEventsSortDescending;
	aToSort : T_LoggedEvents;
	hr		: HRESULT;	
END_VAR
TEST('Should do nothing if only one event received');
// Arrange
aToSort[0].nUniqueId 	:= 1;
aToSort[0].sMessageText := 'First received message is in slot 0';

// Act
hr := fbSUT.Sort(aLoggedEvents:= aToSort);

// Assert
AssertEquals_DINT(Expected:= S_FALSE,
					Actual:= hr,
					Message:= 'Expected HRESULT=S_FALSE');
			
AssertEquals_UDINT(Expected:= 1,
					Actual:= aToSort[0].nUniqueId,
					Message:= 'Expected nUniqueId = 1');
AssertEquals_STRING(Expected:= 'First received message is in slot 0',
					Actual:= aToSort[0].sMessageText,
					Message:= 'Expected first received message');
AssertEquals_UDINT(Expected:= 0,
					Actual:= aToSort[1].nUniqueId,
					Message:= 'Expected nUniqueId = 0');
AssertEquals_STRING(Expected:= '',
					Actual:= aToSort[1].sMessageText,
					Message:= 'Expected empty string');						
TEST_FINISHED();
END_METHOD

METHOD PRIVATE ShouldDoNothingWhenEmpty
VAR_INPUT
END_VAR
VAR_INST
	fbSUT	: FB_LoggedEventsSortDescending;
	aToSort : T_LoggedEvents;
	hr		: HRESULT;	
END_VAR
TEST('Should do nothing if no event');
// Arrange

// Act
hr := fbSUT.Sort(aLoggedEvents:= aToSort);

// Assert
AssertEquals_DINT(Expected:= S_FALSE,
					Actual:= hr,
					Message:= 'Expected HRESULT=S_FALSE');			
TEST_FINISHED();
END_METHOD

METHOD PRIVATE ShouldSortFiveEventsInDescendingOrderSuccessfully
VAR_INPUT
END_VAR
VAR_INST
	fbSUT	: FB_LoggedEventsSortDescending;
	aToSort : T_LoggedEvents;
	hr		: HRESULT;	
END_VAR
TEST('Should sort 5 Items in descending order (newest first)');
// Arrange
aToSort[0].nUniqueId 	:= 1;
aToSort[0].sMessageText := '1st received message was in slot 0';
aToSort[1].nUniqueId 	:= 2;
aToSort[1].sMessageText := '2nd received message was in slot 1';
aToSort[2].nUniqueId 	:= 3;
aToSort[2].sMessageText := '3rd received message was in slot 2';
aToSort[3].nUniqueId 	:= 4;
aToSort[3].sMessageText := '4th received message was in slot 3';
aToSort[4].nUniqueId 	:= 5;
aToSort[4].sMessageText := '5th received message was in slot 4';
// Act
hr := fbSUT.Sort(aLoggedEvents:= aToSort);

// Assert
AssertEquals_DINT(Expected:= S_OK,
					Actual:= hr,
					Message:= 'Expected HRESULT=S_OK');
AssertEquals_UDINT(Expected:= 5,
					Actual:= aToSort[0].nUniqueId,
					Message:= 'Expected nUniqueId = 5');
AssertEquals_STRING(Expected:= '5th received message was in slot 4',
					Actual:= aToSort[0].sMessageText,
					Message:= 'Expected 5th received message');						
AssertEquals_UDINT(Expected:= 4,
					Actual:= aToSort[1].nUniqueId,
					Message:= 'Expected nUniqueId = 4');
AssertEquals_STRING(Expected:= '4th received message was in slot 3',
					Actual:= aToSort[1].sMessageText,
					Message:= 'Expected 4th received message');							
AssertEquals_UDINT(Expected:= 3,
					Actual:= aToSort[2].nUniqueId,
					Message:= 'Expected nUniqueId = 3');
AssertEquals_STRING(Expected:= '3rd received message was in slot 2',
					Actual:= aToSort[2].sMessageText,
					Message:= 'Expected 3rd received message');		
AssertEquals_UDINT(Expected:= 2,
					Actual:= aToSort[3].nUniqueId,
					Message:= 'Expected nUniqueId = 2');
AssertEquals_STRING(Expected:= '2nd received message was in slot 1',
					Actual:= aToSort[3].sMessageText,
					Message:= 'Expected 2nd received message');		
AssertEquals_UDINT(Expected:= 1,
					Actual:= aToSort[4].nUniqueId,
					Message:= 'Expected nUniqueId = 1');
AssertEquals_STRING(Expected:= '1st received message was in slot 0',
					Actual:= aToSort[4].sMessageText,
					Message:= 'Expected 1st received message');		
TEST_FINISHED();
END_METHOD

METHOD PRIVATE ShouldSortFourEventsInDescendingOrderSuccessfully
VAR_INPUT
END_VAR
VAR_INST
	fbSUT	: FB_LoggedEventsSortDescending;
	aToSort : T_LoggedEvents;
	hr		: HRESULT;	
END_VAR
TEST('Should sort 4 Items in descending order (newest first)');
// Arrange
aToSort[0].nUniqueId 	:= 1;
aToSort[0].sMessageText := '1st received message was in slot 0';
aToSort[1].nUniqueId 	:= 2;
aToSort[1].sMessageText := '2nd received message was in slot 1';
aToSort[2].nUniqueId 	:= 3;
aToSort[2].sMessageText := '3rd received message was in slot 2';
aToSort[3].nUniqueId 	:= 4;
aToSort[3].sMessageText := '4th received message was in slot 3';
// Act
hr := fbSUT.Sort(aLoggedEvents:= aToSort);

// Assert
AssertEquals_DINT(Expected:= S_OK,
					Actual:= hr,
					Message:= 'Expected HRESULT=S_OK');
AssertEquals_UDINT(Expected:= 4,
					Actual:= aToSort[0].nUniqueId,
					Message:= 'Expected nUniqueId = 4');
AssertEquals_STRING(Expected:= '4th received message was in slot 3',
					Actual:= aToSort[0].sMessageText,
					Message:= 'Expected 4th received message');							
AssertEquals_UDINT(Expected:= 3,
					Actual:= aToSort[1].nUniqueId,
					Message:= 'Expected nUniqueId = 3');
AssertEquals_STRING(Expected:= '3rd received message was in slot 2',
					Actual:= aToSort[1].sMessageText,
					Message:= 'Expected 3rd received message');		
AssertEquals_UDINT(Expected:= 2,
					Actual:= aToSort[2].nUniqueId,
					Message:= 'Expected nUniqueId = 2');
AssertEquals_STRING(Expected:= '2nd received message was in slot 1',
					Actual:= aToSort[2].sMessageText,
					Message:= 'Expected 2nd received message');		
AssertEquals_UDINT(Expected:= 1,
					Actual:= aToSort[3].nUniqueId,
					Message:= 'Expected nUniqueId = 1');
AssertEquals_STRING(Expected:= '1st received message was in slot 0',
					Actual:= aToSort[3].sMessageText,
					Message:= 'Expected 1st received message');		
TEST_FINISHED();
END_METHOD

METHOD PRIVATE ShouldSortThreeEventsInDescendingOrderSuccessfully
VAR_INPUT
END_VAR
VAR_INST
	fbSUT	: FB_LoggedEventsSortDescending;
	aToSort : T_LoggedEvents;
	hr		: HRESULT;	
END_VAR
TEST('Should sort 3 Items in descending order (newest first)');
// Arrange
aToSort[0].nUniqueId 	:= 1;
aToSort[0].sMessageText := 'First received message was in slot 0';
aToSort[1].nUniqueId 	:= 2;
aToSort[1].sMessageText := 'Second received message was in slot 1';
aToSort[2].nUniqueId 	:= 3;
aToSort[2].sMessageText := 'Third received message was in slot 2';
// Act
hr := fbSUT.Sort(aLoggedEvents:= aToSort);

// Assert
AssertEquals_DINT(Expected:= S_OK,
					Actual:= hr,
					Message:= 'Expected HRESULT=S_OK');
AssertEquals_UDINT(Expected:= 3,
					Actual:= aToSort[0].nUniqueId,
					Message:= 'Expected nUniqueId = 3');
AssertEquals_STRING(Expected:= 'Third received message was in slot 2',
					Actual:= aToSort[0].sMessageText,
					Message:= 'Expected second received message');						
AssertEquals_UDINT(Expected:= 2,
					Actual:= aToSort[1].nUniqueId,
					Message:= 'Expected nUniqueId = 2');
AssertEquals_STRING(Expected:= 'Second received message was in slot 1',
					Actual:= aToSort[1].sMessageText,
					Message:= 'Expected second received message');					
AssertEquals_UDINT(Expected:= 1,
					Actual:= aToSort[2].nUniqueId,
					Message:= 'Expected nUniqueId = 1');
AssertEquals_STRING(Expected:= 'First received message was in slot 0',
					Actual:= aToSort[2].sMessageText,
					Message:= 'Expected first received message');				
TEST_FINISHED();
END_METHOD

METHOD PRIVATE ShouldSortTwoEventsInDescendingOrderSuccessfully
VAR_INPUT
END_VAR
VAR_INST
	fbSUT	: FB_LoggedEventsSortDescending;
	aToSort : T_LoggedEvents;
	hr		: HRESULT;	
END_VAR
TEST('Should sort 2 Items in descending order (newest first)');
// Arrange
aToSort[0].nUniqueId 	:= 1;
aToSort[0].sMessageText := 'First received message was in slot 0';
aToSort[1].nUniqueId 	:= 2;
aToSort[1].sMessageText := 'Second received message was in slot 1';

// Act
hr := fbSUT.Sort(aLoggedEvents:= aToSort);

// Assert
AssertEquals_DINT(Expected:= S_OK,
					Actual:= hr,
					Message:= 'Expected HRESULT=S_OK');
AssertEquals_UDINT(Expected:= 2,
					Actual:= aToSort[0].nUniqueId,
					Message:= 'Expected nUniqueId = 2');
AssertEquals_STRING(Expected:= 'Second received message was in slot 1',
					Actual:= aToSort[0].sMessageText,
					Message:= 'Expected second received message');					
AssertEquals_UDINT(Expected:= 1,
					Actual:= aToSort[1].nUniqueId,
					Message:= 'Expected nUniqueId = 1');
AssertEquals_STRING(Expected:= 'First received message was in slot 0',
					Actual:= aToSort[1].sMessageText,
					Message:= 'Expected first received message');				
TEST_FINISHED();
END_METHOD

METHOD PRIVATE ShouldSortXEventsInDescendingOrderSuccessfully
VAR_INPUT
END_VAR
VAR_INST
	fbSUT	: FB_LoggedEventsSortDescending;
	aToSort : T_LoggedEvents;
	hr		: HRESULT;
	
	i,j 	: UDINT;
	fbFrmt 	: FB_FormatString2;	
	sFrmt 	: STRING := '%d. received message was in slot %d';
	sMsgTxt	: T_MaxString;
END_VAR
VAR CONSTANT
	cUpperBound : UDINT := Param_EventLoggerListener.cMaxConcurrentEvents - 1;
END_VAR
TEST('Should sort X Items in descending order (newest first)');
// Arrange

FOR i:= 0 TO cUpperBound DO
	j := i + 1;
	fbFrmt(
		pFormatString:= ADR(sFrmt), 
		arg1:= F_UDINT(j),
		arg2:= F_UDINT(i), 
		pDstString:= ADR(sMsgTxt), 
		nDstSize:= SIZEOF(sMsgTxt) - 1);
	aToSort[i].nUniqueId 	:= i + 1;
	aToSort[i].sMessageText := sMsgTxt;
END_FOR

// Act
hr := fbSUT.Sort(aLoggedEvents:= aToSort);

// Assert
AssertEquals_DINT(Expected:= S_OK,
					Actual:= hr,
					Message:= 'Expected HRESULT=S_OK');
					
sFrmt := 'Expected nUniqueId = %d';
FOR i:= 0 TO cUpperBound DO
	j:=cUpperBound - i + 1;
	fbFrmt(
		pFormatString:= ADR(sFrmt), 
		arg1:= F_UDINT(j), 
		pDstString:= ADR(sMsgTxt), 
		nDstSize:= SIZEOF(sMsgTxt) - 1);

	AssertEquals_UDINT(Expected:= cUpperBound - i + 1,
					Actual:= aToSort[i].nUniqueId,
					Message:= sMsgTxt);
END_FOR

TEST_FINISHED();
END_METHOD

END_FUNCTION_BLOCK
